# EPICS substitutions: ek9000App/Db/user.substitutions
# Example substitutions file

file "db/dbExample1.db" {
    { user = "jeremy" }
}

file db/dbExample2.db {
    pattern { user, no, scan }
        { "jeremy", 1, "1 second" }
        { "jeremy", 2, "2 second" }
        { "jeremy", 3, "5 second" }
}
